(* Schneider Machine Expert - Basic project Questao3.9_FelipeV1_20241014, file version 2.9.0.0 *)
(* ProjectInformations: Name=Novo projeto *)

HARDWARE
  Cpu 0: TM221M16R/G
  EthernetConfiguration: NetworkName=M221, IpAllocationMode=FixedAddress, IpAddress=0.0.0.0, SubnetMask=0.0.0.0
  SerialLineConfiguration: Baud=Baud19200, Parity=ParityEven, DataBits=DataBits8, StopBits=StopBits1, PhysicalMedium=PhysicalMediumRs485, TransmissionMode=TransmissionModeModbusRtu, SlaveId=1, Addressing=SlaveAddressing
  MastTask: UsePeriodScanMode=false, PeriodScan=100
  FastTask: Period=255
  CpuBehavior: StartingMode=StartAsPreviousState, AutoSaveRamOnEeprom=true, WatchdogPeriod=250

SYMBOLS  (address, symbol, comment, settings)
  %M0       ACIO_BOT
  %M1       PULSO_A
  %M10      AUX_PULSO
  %M11      PULSO_MULT_5
  %M20      LIG_LED_A
  %C0       CONT_PULSO_MULT_5  [Preset=5]
  %I0.0     ATUA_BOTAO
  %Q0.1     LED_A

POU Entrada
  (* SectionNumber=1 *)

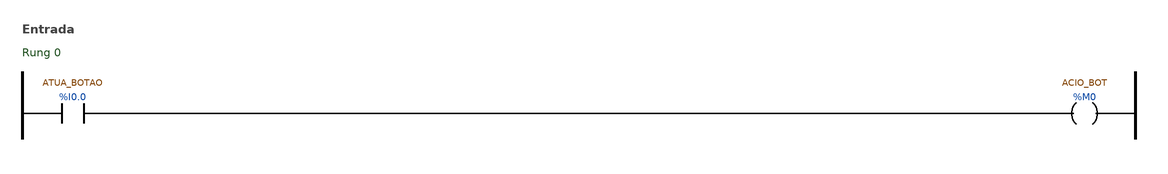

// Rung 0
  LD %I0.0                (* ATUA_BOTAO *)
  ST %M0                  (* ACIO_BOT *)
  // as ST:
  //   ACIO_BOT := ATUA_BOTAO;

POU Lógica
  (* SectionNumber=2 *)

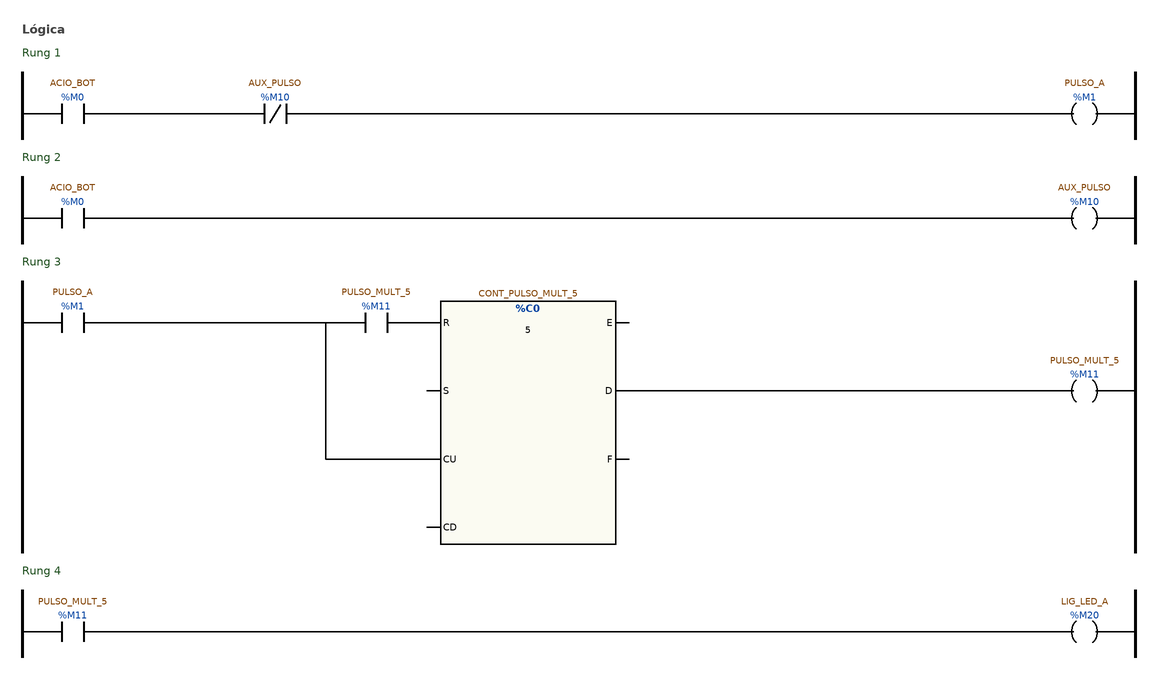

// Rung 1
  LD %M0                  (* ACIO_BOT *)
  ANDN %M10               (* AUX_PULSO *)
  ST %M1                  (* PULSO_A *)
  // as ST:
  //   PULSO_A := ACIO_BOT AND NOT AUX_PULSO;

// Rung 2
  LD %M0                  (* ACIO_BOT *)
  ST %M10                 (* AUX_PULSO *)
  // as ST:
  //   AUX_PULSO := ACIO_BOT;

// Rung 3
  BLK %C0                 (* CONT_PULSO_MULT_5 *)
  LD %M1                  (* PULSO_A *)
  MPS
  AND %M11                (* PULSO_MULT_5 *)
  R
  MPP
  CU
  OUT_BLK
  LD D
  ST %M11                 (* PULSO_MULT_5 *)
  END_BLK
  // as ST:
  //   CONT_PULSO_MULT_5(R := PULSO_A AND PULSO_MULT_5, CU := PULSO_A);
  //   PULSO_MULT_5 := CONT_PULSO_MULT_5.D;

// Rung 4
  LD %M11                 (* PULSO_MULT_5 *)
  ST %M20                 (* LIG_LED_A *)
  // as ST:
  //   LIG_LED_A := PULSO_MULT_5;

POU Saída
  (* SectionNumber=3 *)

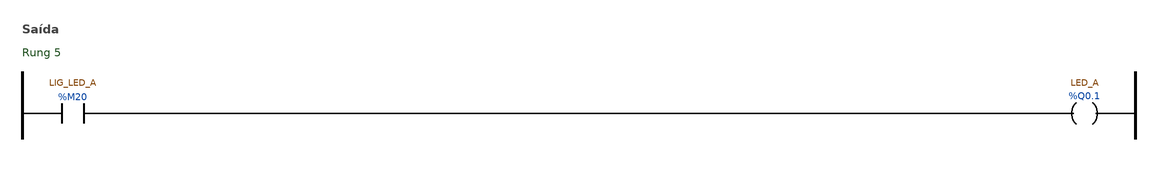

// Rung 5
  LD %M20                 (* LIG_LED_A *)
  ST %Q0.1                (* LED_A *)
  // as ST:
  //   LED_A := LIG_LED_A;
